DATA_BLOCK "DBl_SCALE_CS_1"
{ S7_Optimized_Access := 'FALSE' }
VERSION : 0.1
   STRUCT
      Data { S7_SetPoint := 'False'} : "UDT_SIWA_CS";
   END_STRUCT;


BEGIN

END_DATA_BLOCK

